PROGRAM C_Regul_Temp
VAR
	TON_Chaud: TON;
	TON_Froid: TON;
	Cons_Regul_Chaud: REAL;
	Cons_Regul_Froid: REAL;
	Interdiction_Chaud: BOOL;
	Interdiction_Froid: BOOL;
	Bool_Reg_chaud: BOOL;
	Bool_Reg_froid: BOOL;
	Grad_Cons: UP_DOWN_RATE;
	Calc_Cons_Chaud: REAL;
	Regul_Souf_Chaud: PID;
	Inter_Souf_Chaud: BOOL;
	Regul_Temp_Chaud: OSCAT_BASIC.CTRL_PID;
	Sup_PID_Cd: REAL := 0;
	Regul_Temp_Froid: OSCAT_BASIC.CTRL_PID;
	Sup_PID_Fd: REAL := 0;
	Ecart_TempPiece_Consigne: REAL;
	TOF_Stop: TOF;
	RS_enable: RS;
	Regul_Temp_Amb: OSCAT_BASIC.CTRL_PID;
	Consigne_Soufflage: REAL;
END_VAR
VAR // added by the converter: edge detectors and wires of the graphical bodies
    _w1 : REAL;
    _w2, _w3, _w4 : ANY;
END_VAR

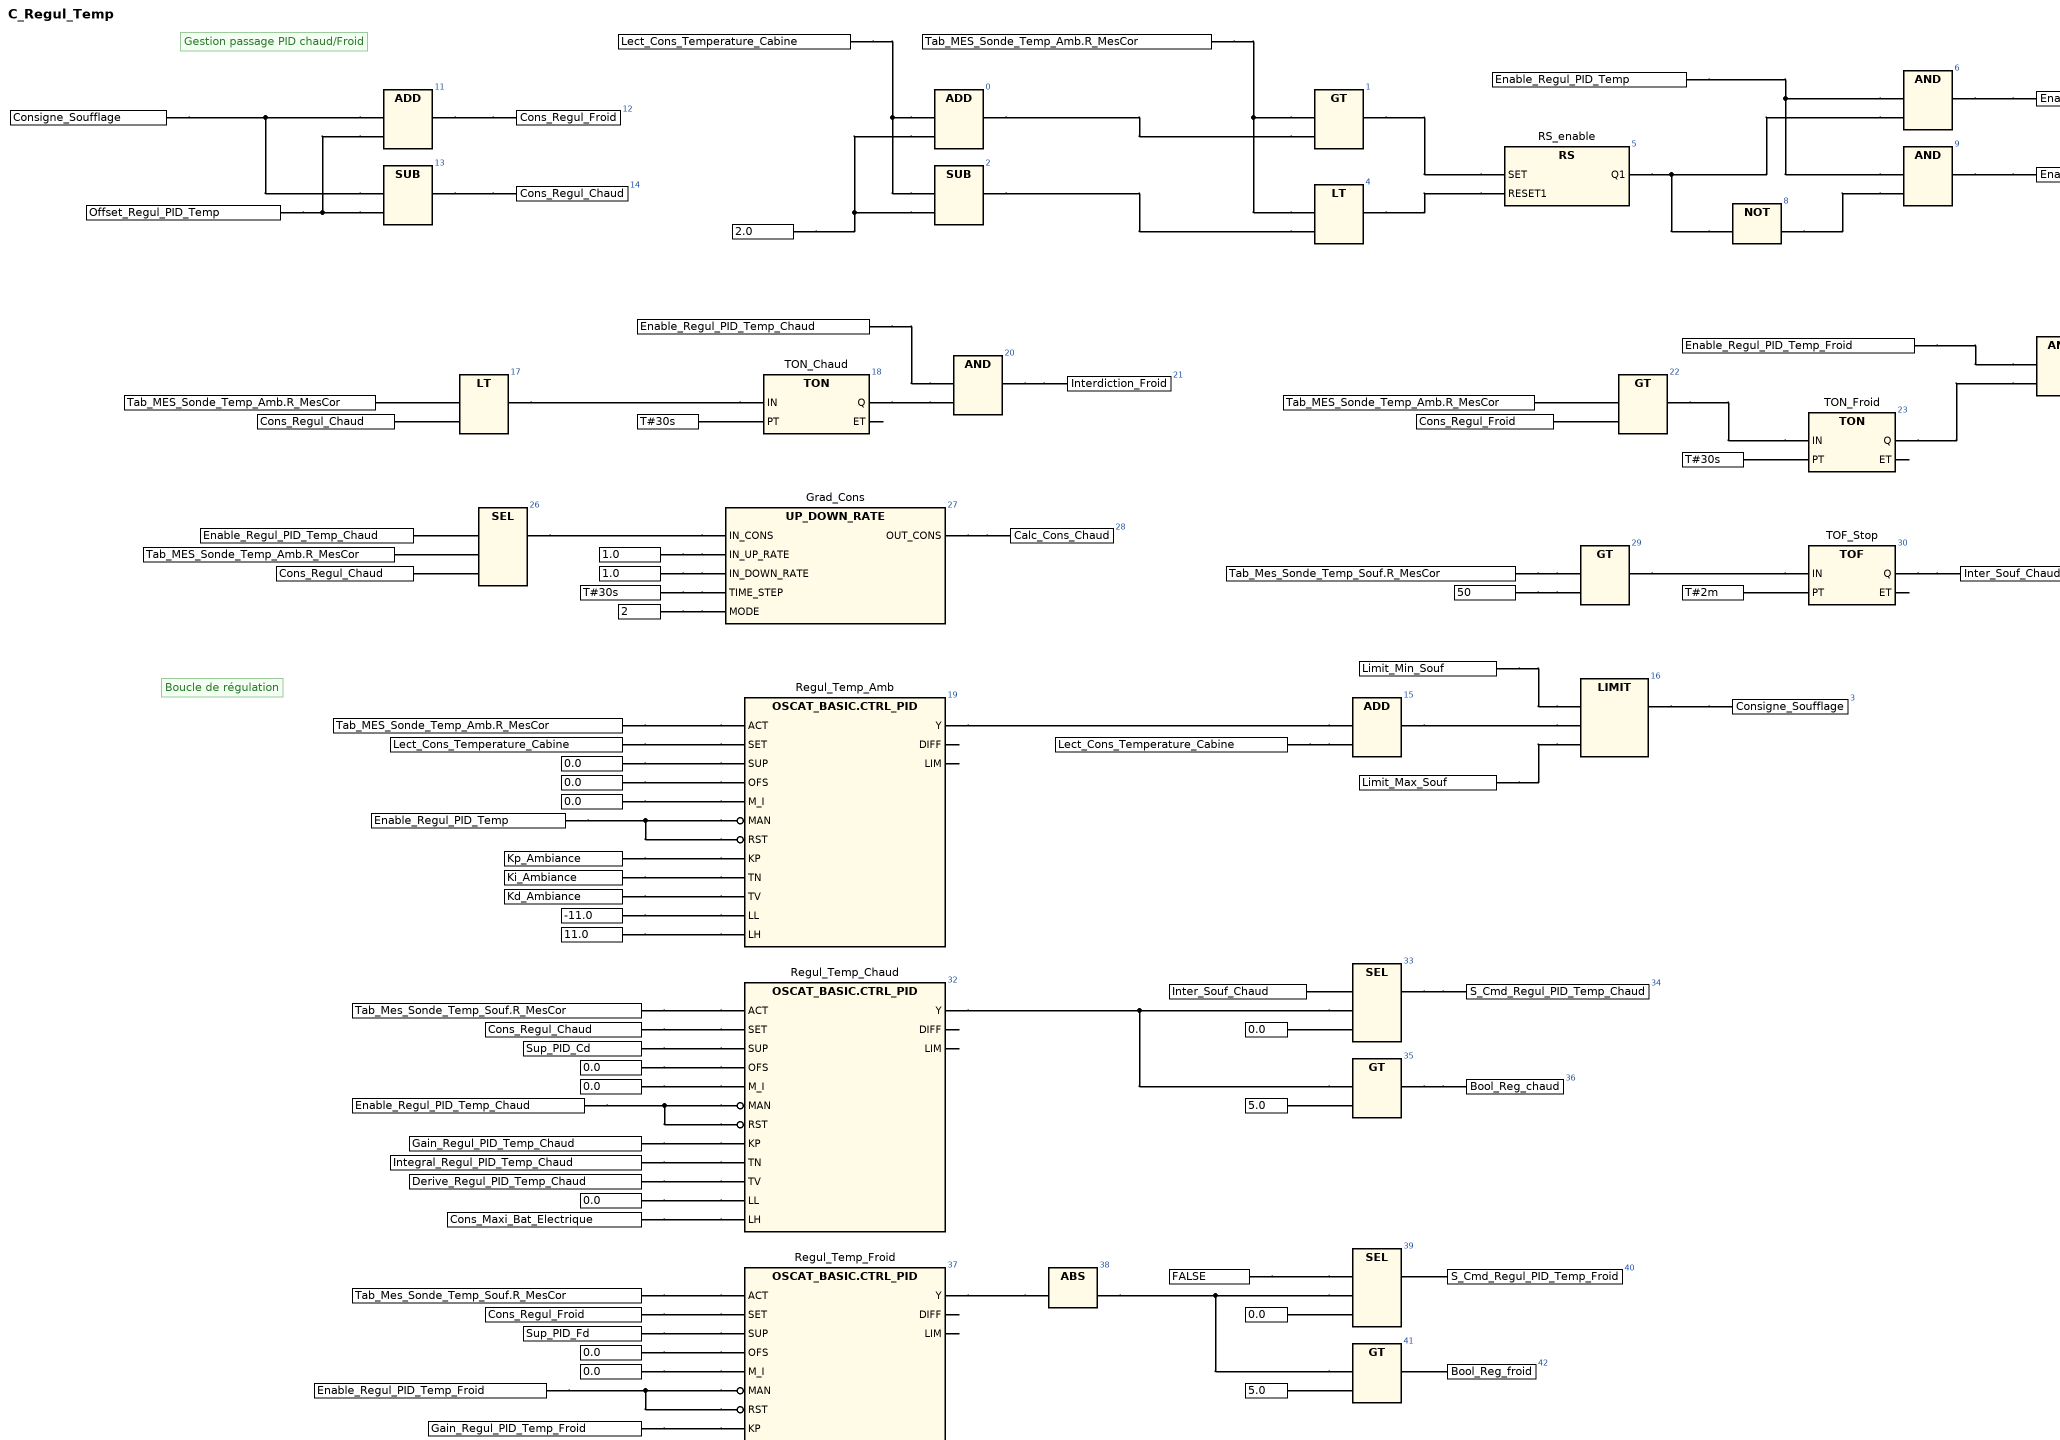
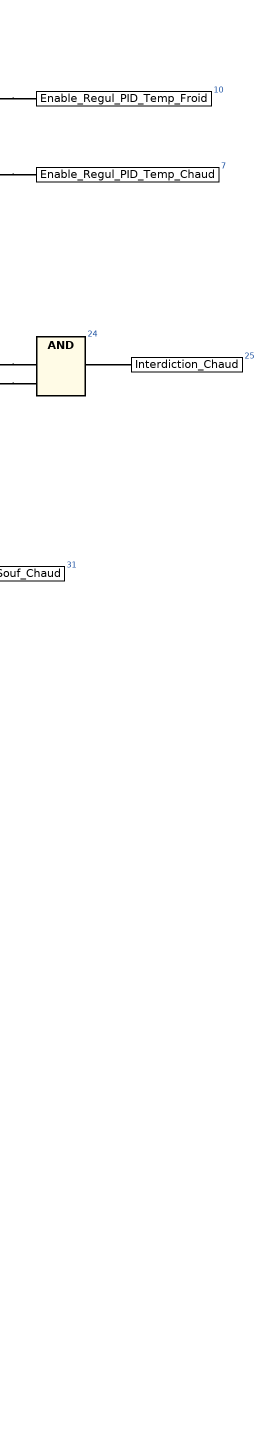
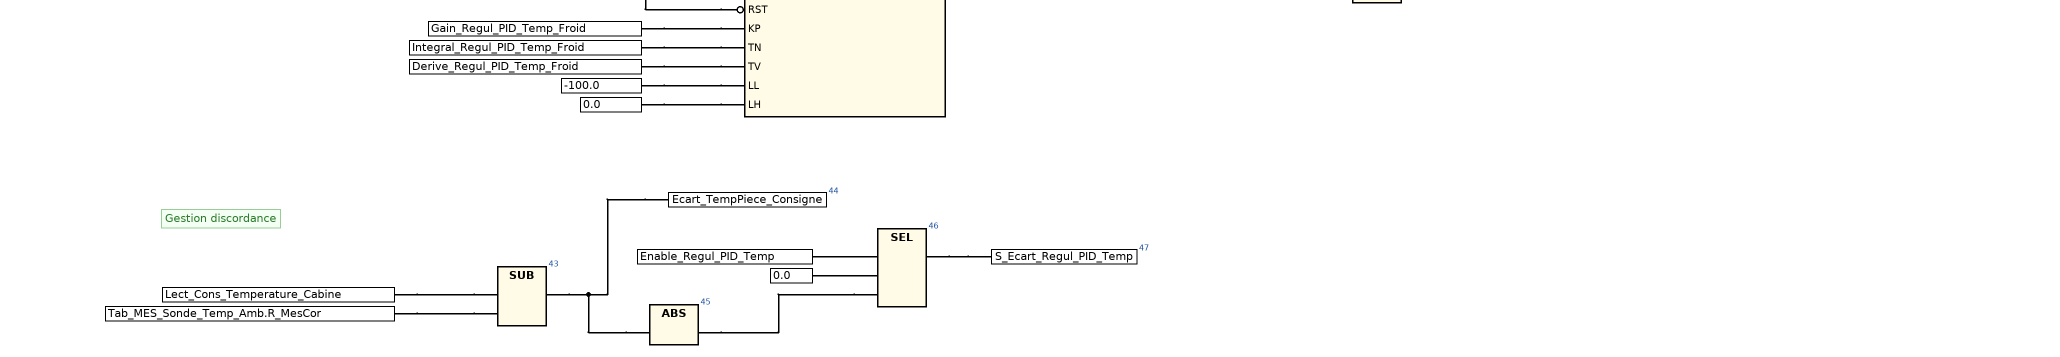
Consigne_Soufflage := _w1;
RS_enable(SET := Tab_MES_Sonde_Temp_Amb.R_MesCor > Lect_Cons_Temperature_Cabine + 2.0, RESET1 := Tab_MES_Sonde_Temp_Amb.R_MesCor < Lect_Cons_Temperature_Cabine - 2.0); // RS
Enable_Regul_PID_Temp_Chaud := _w2;
_w2 := Enable_Regul_PID_Temp AND NOT RS_enable.Q1;
Enable_Regul_PID_Temp_Froid := Enable_Regul_PID_Temp AND RS_enable.Q1;
// Gestion passage PID chaud/Froid
Cons_Regul_Froid := Consigne_Soufflage + Offset_Regul_PID_Temp;
Cons_Regul_Chaud := Consigne_Soufflage - Offset_Regul_PID_Temp;
_w1 := LIMIT(Limit_Min_Souf, Regul_Temp_Amb.Y + Lect_Cons_Temperature_Cabine, Limit_Max_Souf);
TON_Chaud(IN := Tab_MES_Sonde_Temp_Amb.R_MesCor < Cons_Regul_Chaud, PT := T#30s); // TON
// Boucle de régulation
Regul_Temp_Amb(
    ACT := Tab_MES_Sonde_Temp_Amb.R_MesCor,
    SET := Lect_Cons_Temperature_Cabine,
    SUP := 0.0,
    OFS := 0.0,
    M_I := 0.0,
    MAN := NOT Enable_Regul_PID_Temp,
    RST := NOT Enable_Regul_PID_Temp,
    KP := Kp_Ambiance,
    TN := Ki_Ambiance,
    TV := Kd_Ambiance,
    LL := -11.0,
    LH := 11.0); // OSCAT_BASIC.CTRL_PID
Interdiction_Froid := Enable_Regul_PID_Temp_Chaud AND TON_Chaud.Q;
TON_Froid(IN := Tab_MES_Sonde_Temp_Amb.R_MesCor > Cons_Regul_Froid, PT := T#30s); // TON
Interdiction_Chaud := Enable_Regul_PID_Temp_Froid AND TON_Froid.Q;
Grad_Cons(
    IN_CONS := SEL(Enable_Regul_PID_Temp_Chaud, Tab_MES_Sonde_Temp_Amb.R_MesCor, Cons_Regul_Chaud),
    IN_UP_RATE := 1.0,
    IN_DOWN_RATE := 1.0,
    TIME_STEP := T#30s,
    MODE := 2); // UP_DOWN_RATE
Calc_Cons_Chaud := Grad_Cons.OUT_CONS;
TOF_Stop(IN := Tab_Mes_Sonde_Temp_Souf.R_MesCor > 50, PT := T#2m); // TOF
Inter_Souf_Chaud := TOF_Stop.Q;
Regul_Temp_Chaud(
    ACT := Tab_Mes_Sonde_Temp_Souf.R_MesCor,
    SET := Cons_Regul_Chaud,
    SUP := Sup_PID_Cd,
    OFS := 0.0,
    M_I := 0.0,
    MAN := NOT Enable_Regul_PID_Temp_Chaud,
    RST := NOT Enable_Regul_PID_Temp_Chaud,
    KP := Gain_Regul_PID_Temp_Chaud,
    TN := Integral_Regul_PID_Temp_Chaud,
    TV := Derive_Regul_PID_Temp_Chaud,
    LL := 0.0,
    LH := Cons_Maxi_Bat_Electrique); // OSCAT_BASIC.CTRL_PID
S_Cmd_Regul_PID_Temp_Chaud := SEL(Inter_Souf_Chaud, Regul_Temp_Chaud.Y, 0.0);
Bool_Reg_chaud := Regul_Temp_Chaud.Y > 5.0;
Regul_Temp_Froid(
    ACT := Tab_Mes_Sonde_Temp_Souf.R_MesCor,
    SET := Cons_Regul_Froid,
    SUP := Sup_PID_Fd,
    OFS := 0.0,
    M_I := 0.0,
    MAN := NOT Enable_Regul_PID_Temp_Froid,
    RST := NOT Enable_Regul_PID_Temp_Froid,
    KP := Gain_Regul_PID_Temp_Froid,
    TN := Integral_Regul_PID_Temp_Froid,
    TV := Derive_Regul_PID_Temp_Froid,
    LL := -100.0,
    LH := 0.0); // OSCAT_BASIC.CTRL_PID
_w3 := ABS(Regul_Temp_Froid.Y);
S_Cmd_Regul_PID_Temp_Froid := SEL(FALSE, _w3, 0.0);
Bool_Reg_froid := _w3 > 5.0;
// Gestion discordance
_w4 := Lect_Cons_Temperature_Cabine - Tab_MES_Sonde_Temp_Amb.R_MesCor;
Ecart_TempPiece_Consigne := _w4;
S_Ecart_Regul_PID_Temp := SEL(Enable_Regul_PID_Temp, 0.0, ABS(_w4));

END_PROGRAM

(* stored: Version 1.1.0.1, ProductVersion 3.1.4024.16
   POU C_Regul_Temp: Id {0482647d-4fa4-47eb-99d1-edd5e72f46d0}, SpecialFunc None *)
